TYPE ST_HMI_BASE_MODULE_MANUAL_OUT :
STRUCT
	bManualMode			: BOOL;	
	stManualCylinder	: ST_HMI_MANUAL_CYLINDER_OUT;
	stManualDrive		: ST_HMI_MANUAL_DRIVE_OUT;
	stManualAxis		: ST_HMI_MANUAL_AXIS_OUT;
	stManualDevice		: ST_HMI_MANUAL_DEVICE_OUT;
	
	stObjects			: ARRAY[0..iMaxIdxObject] OF ST_Object_Item; // e.g.: fbAxis, ...	
END_STRUCT
END_TYPE

(* stored: Version 1.1.0.1, ProductVersion 3.1.4024.12
   DUT ST_HMI_BASE_MODULE_MANUAL_OUT: Id {979ecc3c-7d84-4c7a-8aa8-7775f65c906b} *)
